(* CODESYS project Server_03.project

Project tree, tasks and I/O mapping:
  Device : CPX-CEC-C1-V3, Festo AG & Co. KG, order no. 3473128, version 3.5.7.30
      unmapped channels: Rotary switch
    application Application
      libraries: Standard, * (System)
      task MainTask (cyclic, interval t#20ms, priority 20) calls PLC_PRG
      program PLC_PRG [LD]
    PLC_Diagnosis : PLC-Diagnosis, Festo AG & Co. KG, version 3.5.4.1
    CPX_System : CPX_System, Festo AG & Co. KG, order no. 3473128, version 1.233
      CEC_C1_V3 : CEC-C1-V3, Festo AG & Co. KG, order no. 3473128, version 1.233
      _8DI_8DO : 8DI/8DO, Festo AG & Co. KG, order no. 526257, version 1.233
          settings:  = 1;  = 1;  = 1;  = 1;  = 0;  = 1;  = 1;  = 0;  = 0;  = 0;  = 0;  = 0;  = 0;  = 0;  = 0;  = 0;  = 0;  = 0;  = 0;  = 0;  = 0;  = 0;  = 0;  = 0;  = 0;  = 0;  = 0;  = 0;  = 0;  = 0;  = 0;  = 0;  = 0;  = 0;  = 0;  = 0;  = 0;  = 0;  = 0;  = 0;
             = 0;  = 0;  = 0;  = 0;  = 0;  = 0;  = 0;  = 0;  = 0;  = 0;  = 0;  = 0;  = 0;  = 0;  = 0;  = 0;  = 0;  = 0;  = 0;  = 0;  = 0;  = 0;  = 0;  = 0;  = 0;  = 0;  = 0;  = 0;  = 0;  = 0;  = 0;  = 0;  = 0;  = 0;  = 0;  = 0;  = 0;  = 0;  = 0;  = 'PI%i.0.0.1=1';
             = 'PI%i.0.1.1=1';  = 'PI%i.0.2.1=1';  = 'PI%i.1.0.1=1';  = 'PI%i.1.1.1=0';  = 'PI%i.1.4.2=1';  = 'PI%i.1.6.2=1';  = 'PI%i.6.0.1=0';  = 'PI%i.6.1.1=0';  = 'PI%i.6.2.1=0';  = 'PI%i.6.3.1=0';  = 'PI%i.6.4.1=0';  = 'PI%i.6.5.1=0';  = 'PI%i.6.6.1=0';  = 'PI%i.6.7.1=0';  = -;  = -
          input  presenca_peca_inicio : BOOL  // Input 0.Bit0
          input  peca_metalica_detectada : BOOL  // Input 0.Bit1
          input  peca_vermelha_detectada : BOOL  // Input 0.Bit2
          input  modulo_desvio1_recuado : BOOL  // Input 0.Bit4
          input  modulo_desvio1_avancado : BOOL  // Input 0.Bit5
          input  modulo_desvio2_recuado : BOOL  // Input 0.Bit6
          input  modulo_desvio2_avancado : BOOL  // Input 0.Bit7
          output esteira : BOOL  // Output 0.Bit0
          output avanco_modulo1 : BOOL  // Output 0.Bit1
          output avanco_modulo2 : BOOL  // Output 0.Bit2
          output avanco_atuador_cilindrico : BOOL  // Output 0.Bit3
          unmapped channels: Input 0, Output 0
      _8DI_8DO_1 : 8DI/8DO, Festo AG & Co. KG, order no. 526257, version 1.233
          unmapped channels: Input 0, Output 0
*)

// Device/Application/PLC_PRG
PROGRAM PLC_PRG
VAR
	presenca_peca_inicioo:BOOL;
	peca_metalica_detectadaa:BOOL;
	peca_vermelha_detectadaa:BOOL;
	modulo_desvio1_recuadoo:BOOL;
	modulo_desvio1_avancadoo:BOOL;
	modulo_desvio2_recuadoo:BOOL;
	modulo_desvio2_avancadoo:BOOL;
	
	esteiraa:BOOL;
	avanco_modulo11:BOOL;
	avanco_modulo22:BOOL;
	avanco_atuador_cilindricoo:BOOL;







END_VAR

// NETWORK 1

END_PROGRAM
